INTERFACE I_AnalogOutput EXTENDS I_Channel

PROPERTY P_Value : LREAL
SET
END_SET
END_PROPERTY

END_INTERFACE

(* stored: Version 1.1.0.1
   Itf I_AnalogOutput: Id {38394b15-c89b-01d7-29f2-baf89f85219c}
   Property P_Value: Id {b9f26c74-154a-0c1d-067b-bd0be1905f18}
   Set Set: Id {41b2dbf6-3383-00bd-3a95-7b759629dfb1} *)
